Fanuc KAREL source: ko00002.KL

PROGRAM KO00002
%STACKSIZE=65535
%PRIORITY=65535
%NOLOCKGROUP
VAR
P1 : POSITION
P2 : POSITION
P3 : POSITION
OUT : XYZWPR
BEGIN
-- UNRESOLVED_PC line 9 opcodes [27 22 1C 22 1C 22 1C 76 7E 4A] marker_code=0
END KO00002
